(* CODESYS project Modbus_RTU_UART.project

Project tree, tasks and I/O mapping:
  Device : CODESYS Control for Raspberry Pi, 3S - Smart Software Solutions GmbH, version 3.5.8.10
    application Application
      libraries: Standard, * (System); Raspberry SPI MCP3008, 1.1.0.0 (3S - Smart Software Solutions GmbH); Util, * (System)
      task MainTask (cyclic, interval t#20ms, priority 1) calls PLC_PRG
      task VISU_TASK (cyclic, interval 100 ms, priority 31) calls VisuElems.Visu_Prg
      task Termosensors (cyclic, interval t#1000ms, priority 13) calls Termosensors
      program PLC_PRG [ST]
      visualisation Modbus
      program Termosensors [ST]
    SoftMotion General Axis Pool
    GPIOs_A_B : GPIOs B+/Pi2, 3S - Smart Software Solutions GmbH, version 1.1.1.10
        output Application.PLC_PRG.out_1 : BOOL  // digital outputs (GPIO0..GPIO31).Bit17
        output Application.PLC_PRG.out_3 : BOOL  // digital outputs (GPIO0..GPIO31).Bit27
        unmapped channels: digital inputs (GPIO0..GPIO31), digital outputs (GPIO0..GPIO31)
    I²C
    SPI
    Onewire
      Onewire_master : Onewire master, 3S - Smart Software Solutions GmbH, version 1.0.0.0
        DS18B20 : DS18B20, 3S - Smart Software Solutions GmbH, version 1.3.0.0
            settings: Unique device address = '28-000005b29557'
        DS18B20_1 : DS18B20, 3S - Smart Software Solutions GmbH, version 1.3.0.0
            settings: Unique device address = '28-0000066e2bd4'
    Camera device
      <Empty>
    Modbus_COM : Modbus COM, 3S - Smart Software Solutions GmbH, version 3.4.0.0
        settings: DataBits = 8; StopBits = 1; ComPort = 1
      Modbus_Master_COM_Port : Modbus Master, COM Port, 3S - Smart Software Solutions GmbH, version 3.5.5.0
          settings: Transmission = 'RTU'; ResponseTimeout = 1000; TimeBetweenFrames = 10; Auto-restart communication = TRUE
        Modbus_Slave_COM_Port : Modbus Slave, COM Port, 3S - Smart Software Solutions GmbH, version 3.5.4.0
            settings: status.Function Code = 3; status.Read Offset = 16#2100; status.Read Length = 1; status.Write Offset = 0; status.Write Length = 0; status.Cycle Time = 100; frequency.Function Code = 3; frequency.Read Offset = 16#1101; frequency.Read Length = 1; frequency.Write Offset = 0; frequency.Write Length = 0; frequency.Cycle Time = 100; voltage.Function Code = 3; voltage.Read Offset = 16#3002; voltage.Read Length = 1; voltage.Write Offset = 0; voltage.Write Length = 0; voltage.Cycle Time = 100; current.Function Code = 3; current.Read Offset = 16#3004; current.Read Length = 1; current.Write Offset = 0; current.Write Length = 0; current.Cycle Time = 100; speed.Function Code = 3; speed.Read Offset = 16#3005; speed.Read Length = 1; speed.Write Offset = 0; speed.Write Length = 0; speed.Cycle Time = 100; power.Function Code = 3; power.Read Offset = 16#3006; power.Read Length = 1; power.Write Offset = 0; power.Write Length = 0; power.Cycle Time = 100; torque.Function Code = 3; torque.Read Offset = 16#3007; torque.Read Length = 1; torque.Write Offset = 0;
              torque.Write Length = 0; torque.Cycle Time = 100; control_mb.Function Code = 6; control_mb.Read Offset = 0; control_mb.Read Length = 0; control_mb.Write Offset = 16#2000; control_mb.Write Length = 1; control_mb.Cycle Time = 100; Otput_voltage.Function Code = 3; Otput_voltage.Read Offset = 16#3003; Otput_voltage.Read Length = 1; Otput_voltage.Write Offset = 0; Otput_voltage.Write Length = 0; Otput_voltage.Cycle Time = 100
            input  Application.PLC_PRG.status : WORD  // status.status
            input  Application.PLC_PRG.frequency : WORD  // frequency.frequency
            input  Application.PLC_PRG.voltage : WORD  // voltage.voltage
            input  Application.PLC_PRG.current : WORD  // current.current
            input  Application.PLC_PRG.speed : WORD  // speed.speed
            input  Application.PLC_PRG.power : WORD  // power.power
            input  Application.PLC_PRG.torque : WORD  // torque.torque
            output Application.PLC_PRG.commandToModbus : WORD  // control_mb.control_mb
            input  Application.PLC_PRG.out_voltage : WORD  // Otput_voltage.Otput_voltage
            unmapped channels: status, frequency, voltage, current, speed, power, torque, control_mb, Otput_voltage
  text list GlobalTextList
  GlobalImagePool
  5ce3da45-db07-42e7-a21c-a00fff4ed8f6|wallpapers_25719.jpg
  5ce3da45-db07-42e7-a21c-a00fff4ed8f6|1.jpg
*)

// Device/Application/PLC_PRG
PROGRAM PLC_PRG
VAR
	status,commandToModbus,frequency,voltage,current,speed, power, out_voltage, torque: WORD;
	start,lampOut, out_1, out_3: BOOL;
	freq, volt, volt1: REAL;
	out_gen: BLINK; // библиотека Utils;
	text: STRING;
END_VAR

freq:=WORD_TO_REAL(frequency)/100; // переводим байты в плав.точку и делим на 100, что бы было 50.00;
volt:=WORD_TO_REAL(voltage)/10;    // переводим байты в плав.точку и делим на 10, что бы было xxx,x;
IF start = 1 THEN commandToModbus:=1; // Включаем переключатель и пишем команду пуск в Modbus;
	ELSE commandToModbus:=5;
END_IF

IF status = 1 THEN lampOut:=1; out_1:=1; out_gen(ENABLE:= 1, TIMELOW:=T#0.5S , TIMEHIGH:=T#0.5S , OUT => out_3 ); // мигаем LED;
	ELSE lampOut:=0; out_1:=0; out_3:=0; ; // выключаем все;
END_IF

IF status = 1 THEN text:='RUN';  // Выводим текст статуса инвертора;
	//ELSE text:=' ';  
		IF status=3 THEN text:='STOP';
	END_IF
END_IF

IF status = 2 THEN text:='Reverse';
IF status=3 THEN text:='STOP';
	END_IF
	END_IF

END_PROGRAM

// Device/Application/Termosensors
PROGRAM Termosensors
VAR
astrID: ARRAY[1..20] OF STRING; // касается опроса DS18B20;
	ui: uINT;
	x: BOOL;
	ds_temp: REAL; // регистр температуры 1;
	ds_temp1: REAL; // регистр температуры 2;
END_VAR

IF NOT x THEN
	x := TRUE;
	//scan function
	FOR ui:=1 TO MIN(Onewire_master.uiScannedDevices, 20) DO
		astrID[ui] := Onewire_master.pasScannedDevices^[ui-1].StringRepresentation;
	END_FOR
END_IF

// Выводим значение;
ds_temp:=DS18B20_1.rTemp;
ds_temp1:=DS18B20_1_1.rTemp;

END_PROGRAM

// Device/Application/Modbus
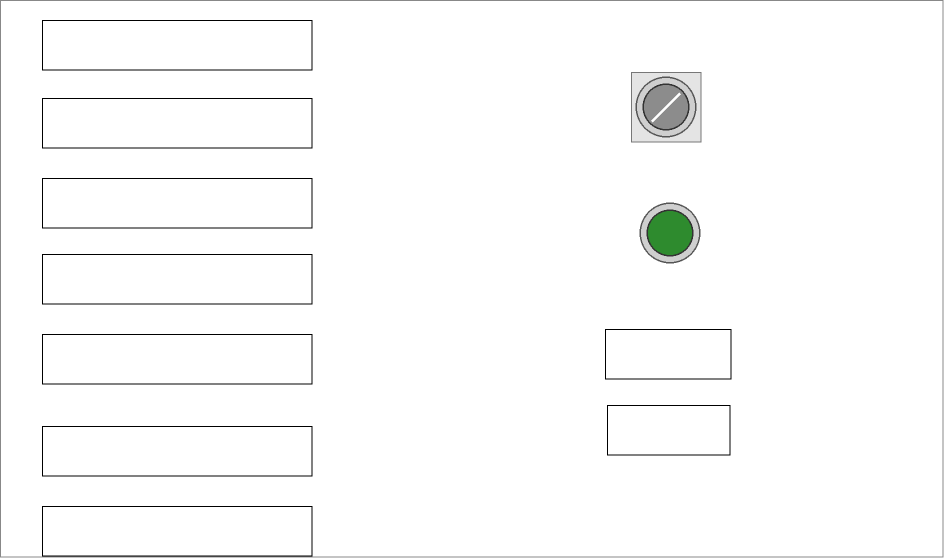
VISUALIZATION Modbus  // 944x558, background image 1
    Lamp1 (635,198 70x70), variable: PLC_PRG.lampOut, style: Lamp-Lamp1-Green
    RotarySwitch (631,72 70x70), variable: PLC_PRG.start, behaviour: TOGGLE, style: Switch-RotarySwitch-Gray
    Rectangle (42,20 270x50), "%s", text variable: PLC_PRG.text
    Rectangle (42,98 270x50), "%s", text variable: PLC_PRG.freq
    Rectangle (42,178 270x50), "%s", text variable: PLC_PRG.volt
    Rectangle (42,334 270x50), "%s", text variable: PLC_PRG.current
    Rectangle (42,426 270x50), "%s", text variable: PLC_PRG.speed
    Rectangle (42,506 270x50), "%s", text variable: PLC_PRG.power
    Rectangle (42,254 270x50), "%s", text variable: PLC_PRG.volt1
    Label (369,107 150x30), "Frequency, Hz"
    Label (369,31 150x29), "Status"
    Label (369,188 150x30), "Bus voltage, V"
    Label (360,347 169x30), "Output current, A"
    Label (369,435 150x30), "Speed, rpm"
    Label (563,34 79x29), "Start"
    Label (679,34 79x29), "Stop"
    Label (624,160 79x29), "Run"
    Label (369,512 150x30), "Power, Wt"
    Label (356,256 177x30), "Output voltage, V"
    Rectangle (605,329 126x50), "%s", text variable: Termosensors.ds_temp
    Rectangle (607,405 123x50), "%s", text variable: Termosensors.ds_temp1
    Label (747,329 195x57), "Indoor temperature, C"
    Label (747,394 195x57), "Outdoor temperature, C"
END_VISUALIZATION
